{attribute 'GeneratedUsingTerminal: ELM3704-0000-0016'}
{attribute addProperty BoxType "ELM3704-0000-0016"}
{attribute addProperty Id "PAI_Status_Channel_1AT %I*PAI_Status_Channel_AE4AC1047PAI_Samples_1_Channel_1AT %I*PAI_Samples_1_Channel_EEA517254PAI_Timestamp_Channel_1AT %I*PAI_Timestamp_Channel_6DC4D2968PAI_Status_Channel_2AT %I*PAI_Status_Channel_AE4AC1047PAI_Samples_1_Channel_2AT %I*PAI_Samples_1_Channel_EEA517254PAI_Status_Channel_3AT %I*PAI_Status_Channel_AE4AC1047PAI_Samples_1_Channel_3AT %I*PAI_Samples_1_Channel_EEA517254PAI_Status_Channel_4AT %I*PAI_Status_Channel_AE4AC1047PAI_Samples_1_Channel_4AT %I*PAI_Samples_1_Channel_EEA517254WcStateAT %I*WcState_9091E0EB2InfoDataAT %I*InfoData_1088C70510"}
{attribute addProperty CRC "394098388"}
{attribute addProperty Size "64"}
TYPE ELM3704_177D76D4 EXTENDS EtcSlaveTerminalBase_947E5A46 :
STRUCT
	{attribute addProperty Name "PAI_Status_Channel_1"}
	PAI_Status_Channel_1 : PAI_Status_Channel_AE4AC104;
	{attribute addProperty Name "PAI_Samples_1_Channel_1"}
	PAI_Samples_1_Channel_1 : PAI_Samples_1_Channel_EEA51725;
	{attribute addProperty Name "PAI_Timestamp_Channel_1"}
	PAI_Timestamp_Channel_1 : PAI_Timestamp_Channel_6DC4D296;
	{attribute addProperty Name "PAI_Status_Channel_2"}
	PAI_Status_Channel_2 : PAI_Status_Channel_AE4AC104;
	{attribute addProperty Name "PAI_Samples_1_Channel_2"}
	PAI_Samples_1_Channel_2 : PAI_Samples_1_Channel_EEA51725;
	{attribute addProperty Name "PAI_Status_Channel_3"}
	PAI_Status_Channel_3 : PAI_Status_Channel_AE4AC104;
	{attribute addProperty Name "PAI_Samples_1_Channel_3"}
	PAI_Samples_1_Channel_3 : PAI_Samples_1_Channel_EEA51725;
	{attribute addProperty Name "PAI_Status_Channel_4"}
	PAI_Status_Channel_4 : PAI_Status_Channel_AE4AC104;
	{attribute addProperty Name "PAI_Samples_1_Channel_4"}
	PAI_Samples_1_Channel_4 : PAI_Samples_1_Channel_EEA51725;
	{attribute addProperty Name "WcState"}
	WcState : WcState_9091E0EB;
	{attribute addProperty Name "InfoData"}
	InfoData : InfoData_1088C705;
END_STRUCT
END_TYPE

(* stored: Version 1.2.0.0, ProductVersion 3.1.4024.9
   DUT ELM3704_177D76D4: Id {921a5149-ba97-4895-a23f-95b2365d23f2} *)
